{attribute 'qualified_only'}
{attribute 'strict'}
TYPE UnitOperation :
(
	NormalOperation := 0, AlwaysStart
);
END_TYPE

(* stored: Version 1.1.0.1, ProductVersion 3.1.4024.6
   DUT UnitOperation: Id {ea3d12ac-7bef-4039-a499-3d1e58013a54} *)
